{attribute addProperty BoxType "EPP2316-0003-0016"}
{attribute addProperty Id "DIG_InputsAT %I*DIG_Inputs_9F71B9E27290DIG_Diag_InputsAT %I*DIG_Diag_Inputs_AC4A9AF06480DIG_Inputs_DeviceAT %I*DIG_Inputs_Device_30BACB404050DIG_OutputsAT %Q*DIG_Outputs_33B763766480DIG_Outputs_DeviceAT %Q*DIG_Outputs_Device_735003021620WcStateAT %I*WcState_F855686C1620InfoDataAT %I*InfoData_BC63D37F80100"}
{attribute addProperty CRC "594889051"}
{attribute addProperty SizeInBites "352"}
{attribute addProperty SizeInBytes "44"}
TYPE EPP2316_91349AC4 :
STRUCT
	{attribute addProperty Name "DIG_Inputs"}
	DIG_Inputs : DIG_Inputs_9F71B9E2;
	{attribute addProperty Name "DIG_Diag_Inputs"}
	DIG_Diag_Inputs : DIG_Diag_Inputs_AC4A9AF0;
	{attribute addProperty Name "DIG_Inputs_Device"}
	DIG_Inputs_Device : DIG_Inputs_Device_30BACB40;
	{attribute addProperty Name "DIG_Outputs"}
	DIG_Outputs : DIG_Outputs_33B76376;
	{attribute addProperty Name "DIG_Outputs_Device"}
	DIG_Outputs_Device : DIG_Outputs_Device_73500302;
	{attribute addProperty Name "WcState"}
	WcState : WcState_F855686C;
	{attribute addProperty Name "InfoData"}
	InfoData : InfoData_BC63D37F;
END_STRUCT
END_TYPE

(* stored: Version 1.2.0.0, ProductVersion 3.1.4024.9
   DUT EPP2316_91349AC4: Id {9a52f3ac-4aac-49b2-9d52-d0f591af64b8} *)
